(* PLC project Adressering.ecp, WAGO e!COCKPIT e!COCKPIT *)
(* stored: creationDateTime 2021-01-18T14:20:23.2110188, modificationDateTime 2021-01-18T11:51:27.6823754 *)

{attribute 'qualified_only'}
VAR_GLOBAL  (* STLV80_563 *)
  STLV80_A_563_5A201 : dtRomtype_1;  (* Gang *)
  STLV80_A_563_5A202 : dtRomtype_11;  (* gang *)
  STLV80_A_563_5A203 : dtRomtype_111;  (* rom *)
  STLV80_A_563_5A301 : dtRomtype_1111;  (* rom2 *)
  STLV80_A_563_5A302 : dtRomtype_11111;  (* rom3 *)
  STLV80_A_563_5B201 : dtRomtype_111111;  (* rom4 *)
  STLV80_A_563_5B202 : dtRomtype_1111111;  (* rom5 *)
  STLV80_A_563_5B301 : dtRomtype_11111111;  (* rom6 *)
  STLV80_A_563_5B302 : dtRomtype_1111111111;  (* rom7 *)
  STLV80_A_563_5C201 : dtRomtype_1100000001;  (* rom8 *)
  STLV80_A_563_5C202 : dtRomtype_1100000010;  (* 1100000010 *)
END_VAR

PROGRAM PRG_563_KNX
  VAR
    i : INT := 0;  (* Felles *)
    Interval : OSCAT_BASIC.CLK_PRG;
    typDPT : typDPT;
    M1_001_5A201_RB601_V : fbDPT_Switch_pro;  (* 5A201 *)
    M1_002_5A202_RB601_V : fbDPT_Switch_pro;  (* 5A202 *)
    M1_003_5A202_RB601_HVAC : fbDPT_Switch_pro;  (* 5A202 *)
    M1_004_5A203_RB601_V : fbDPT_Switch_pro;  (* 5A203 *)
    M1_005_5A203_RB601_HVAC : fbDPT_Switch_pro;  (* 5A203 *)
    M1_006_5A203_RT601_CT : fbDPT_Value_Temp_pro;  (* 5A203 *)
    M1_007_5A301_RB601_V : fbDPT_Switch_pro;  (* 5A301 *)
    M1_008_5A301_RB601_HVAC : fbDPT_Switch_pro;  (* 5A301 *)
    M1_009_5A301_RT601_CT : fbDPT_Value_Temp_pro;  (* 5A301 *)
    M1_010_5A301_RY601_CV : fbDPT_Value_AirQuality_pro;  (* 5A301 *)
    M1_011_5A302_RB601_V : fbDPT_Switch_pro;  (* 5A302 *)
    M1_012_5A302_RB601_HVAC : fbDPT_Switch_pro;  (* 5A302 *)
    M1_013_5A302_RT601_CT : fbDPT_Value_Temp_pro;  (* 5A302 *)
    M1_014_5A302_RY601_CV : fbDPT_Value_AirQuality_pro;  (* 5A302 *)
    M1_015_5A302_LH601_OP : fbDPT_Scaling_pro;  (* 5A302 *)
    M1_016_5B201_RB601_V : fbDPT_Switch_pro;  (* 5B201 *)
    M1_017_5B201_RB601_HVAC : fbDPT_Switch_pro;  (* 5B201 *)
    M1_018_5B201_RT601_CT : fbDPT_Value_Temp_pro;  (* 5B201 *)
    M1_019_5B201_RY601_CV : fbDPT_Value_AirQuality_pro;  (* 5B201 *)
    M1_020_5B201_LH601_OP : fbDPT_Scaling_pro;  (* 5B201 *)
    M1_021_5B201_LH601_CMD : fbDPT_Switch_pro;  (* 5B201 *)
    M1_022_5B202_RB601_V : fbDPT_Switch_pro;  (* 5B202 *)
    M1_023_5B202_RB601_HVAC : fbDPT_Switch_pro;  (* 5B202 *)
    M1_024_5B202_RT601_CT : fbDPT_Value_Temp_pro;  (* 5B202 *)
    M1_025_5B202_RY601_CV : fbDPT_Value_AirQuality_pro;  (* 5B202 *)
    M1_026_5B202_LH601_OP : fbDPT_Scaling_pro;  (* 5B202 *)
    M1_027_5B202_LH601_CMD : fbDPT_Switch_pro;  (* 5B202 *)
    M1_028_5B202_LC601_OP : fbDPT_Scaling_pro;  (* 5B202 *)
    M1_029_5B301_RB601_V : fbDPT_Switch_pro;  (* 5B301 *)
    M1_030_5B301_RB601_HVAC : fbDPT_Switch_pro;  (* 5B301 *)
    M1_031_5B301_RT601_CT : fbDPT_Value_Temp_pro;  (* 5B301 *)
    M1_032_5B301_RY601_CV : fbDPT_Value_AirQuality_pro;  (* 5B301 *)
    M1_033_5B301_LH601_OP : fbDPT_Scaling_pro;  (* 5B301 *)
    M1_034_5B301_LH601_CMD : fbDPT_Switch_pro;  (* 5B301 *)
    M1_035_5B301_LC601_OP : fbDPT_Scaling_pro;  (* 5B301 *)
    M1_036_5B301_LC601_CMD : fbDPT_Switch_pro;  (* 5B301 *)
    M1_037_5B302_RB601_V : fbDPT_Switch_pro;  (* 5B302 *)
    M1_038_5B302_RB601_HVAC : fbDPT_Switch_pro;  (* 5B302 *)
    M1_039_5B302_RT601_CT : fbDPT_Value_Temp_pro;  (* 5B302 *)
    M1_040_5B302_RY601_CV : fbDPT_Value_AirQuality_pro;  (* 5B302 *)
    M1_041_5B302_LH601_OP : fbDPT_Scaling_pro;  (* 5B302 *)
    M1_042_5B302_LH601_CMD : fbDPT_Switch_pro;  (* 5B302 *)
    M1_043_5B302_LC601_OP : fbDPT_Scaling_pro;  (* 5B302 *)
    M1_044_5B302_LC601_CMD : fbDPT_Switch_pro;  (* 5B302 *)
    M1_045_5B302_RT601_SP_FB : fbDPT_Value_Temp_pro;  (* 5B302 *)
    M1_046_5B302_RT601_SP : fbDPT_Value_Temp_pro;  (* 5B302 *)
    M1_047_5C201_RB601_V : fbDPT_Switch_pro;  (* 5C201 *)
    M1_048_5C201_RB601_HVAC : fbDPT_Switch_pro;  (* 5C201 *)
    M1_049_5C201_RT601_SP : fbDPT_Value_Temp_pro;  (* 5C201 *)
    M1_050_5C202_RB601_V : fbDPT_Switch_pro;  (* 5C202 *)
    M1_051_5C202_RB601_HVAC : fbDPT_Switch_pro;  (* 5C202 *)
    M1_052_5C202_RT601_SP_FB : fbDPT_Value_Temp_pro;  (* 5C202 *)
  END_VAR
  VAR  (* added by the conversion: wires and edge detectors of the diagram *)
    _ADD9_OUT : INT;
    _GT15_OUT : BOOL;
    _MOVE19_ENO : BOOL;
    _MOVE19_OUT : INT;
  END_VAR

(* CFC diagram, written out as Structured Text *)
(* KNX Sending interval *)
Interval(PT := t#2M);
_ADD9_OUT := BOOL_TO_INT(Interval.Q) + i;
i := _ADD9_OUT;
_GT15_OUT := i > 13;
_MOVE19_OUT := MOVE(EN := _GT15_OUT, IN := 0, ENO => _MOVE19_ENO);
IF _MOVE19_ENO THEN i := _MOVE19_OUT; END_IF;
(* Rom 5A201 *)
(* RB601_V *)
M1_001_5A201_RB601_V(bPortKNX := 1, dwIndex_DPT := 1, typDPT := typDPT);
STLV80_563.STLV80_A_563_5A201.RB601_V := M1_001_5A201_RB601_V.xSwitch_OUT;
(* Rom 5A202 *)
(* RB601_V *)
(* RB601_HVAC *)
M1_002_5A202_RB601_V(bPortKNX := 1, dwIndex_DPT := 2, typDPT := typDPT);
STLV80_563.STLV80_A_563_5A202.RB601_V := M1_002_5A202_RB601_V.xSwitch_OUT;
M1_003_5A202_RB601_HVAC(bPortKNX := 1, dwIndex_DPT := 3, typDPT := typDPT);
STLV80_563.STLV80_A_563_5A202.RB601_HVAC := M1_003_5A202_RB601_HVAC.xSwitch_OUT;
(* Rom 5A203 *)
(* RB601_V *)
(* RB601_HVAC *)
M1_004_5A203_RB601_V(bPortKNX := 1, dwIndex_DPT := 4, typDPT := typDPT);
STLV80_563.STLV80_A_563_5A203.RB601_V := M1_004_5A203_RB601_V.xSwitch_OUT;
M1_005_5A203_RB601_HVAC(bPortKNX := 1, dwIndex_DPT := 5, typDPT := typDPT);
STLV80_563.STLV80_A_563_5A203.RB601_HVAC := M1_005_5A203_RB601_HVAC.xSwitch_OUT;
(* RT601_CT *)
M1_006_5A203_RT601_CT(bPortKNX := 1, dwIndex_DPT := 6, typDPT := typDPT);
STLV80_563.STLV80_A_563_5A203.RT601_CT := M1_006_5A203_RT601_CT.rValue_OUT;
(* Rom 5A301 *)
(* RB601_V *)
(* RB601_HVAC *)
M1_007_5A301_RB601_V(bPortKNX := 1, dwIndex_DPT := 7, typDPT := typDPT);
STLV80_563.STLV80_A_563_5A301.RB601_V := M1_007_5A301_RB601_V.xSwitch_OUT;
M1_008_5A301_RB601_HVAC(bPortKNX := 1, dwIndex_DPT := 8, typDPT := typDPT);
STLV80_563.STLV80_A_563_5A301.RB601_HVAC := M1_008_5A301_RB601_HVAC.xSwitch_OUT;
(* RT601_CT *)
(* RY601_CV *)
M1_009_5A301_RT601_CT(bPortKNX := 1, dwIndex_DPT := 9, typDPT := typDPT);
STLV80_563.STLV80_A_563_5A301.RT601_CT := M1_009_5A301_RT601_CT.rValue_OUT;
M1_010_5A301_RY601_CV(bPortKNX := 1, dwIndex_DPT := 10, typDPT := typDPT);
STLV80_563.STLV80_A_563_5A301.RY601_CV := M1_010_5A301_RY601_CV.rValue_OUT;
(* Rom 5A302 *)
(* RB601_V *)
(* RB601_HVAC *)
M1_011_5A302_RB601_V(bPortKNX := 1, dwIndex_DPT := 11, typDPT := typDPT);
STLV80_563.STLV80_A_563_5A302.RB601_V := M1_011_5A302_RB601_V.xSwitch_OUT;
M1_012_5A302_RB601_HVAC(bPortKNX := 1, dwIndex_DPT := 12, typDPT := typDPT);
STLV80_563.STLV80_A_563_5A302.RB601_HVAC := M1_012_5A302_RB601_HVAC.xSwitch_OUT;
(* RT601_CT *)
(* RY601_CV *)
M1_013_5A302_RT601_CT(bPortKNX := 1, dwIndex_DPT := 13, typDPT := typDPT);
STLV80_563.STLV80_A_563_5A302.RT601_CT := M1_013_5A302_RT601_CT.rValue_OUT;
M1_014_5A302_RY601_CV(bPortKNX := 1, dwIndex_DPT := 14, typDPT := typDPT);
STLV80_563.STLV80_A_563_5A302.RY601_CV := M1_014_5A302_RY601_CV.rValue_OUT;
(* LH601_OP *)
M1_015_5A302_LH601_OP(bPortKNX := 1, dwIndex_DPT := 15, rValue_IN := STLV80_563.STLV80_A_563_5A302.LH601_OP, xUpdate_KNX := i = 0, typDPT := typDPT);
(* Rom 5B201 *)
(* RB601_V *)
(* RB601_HVAC *)
M1_016_5B201_RB601_V(bPortKNX := 1, dwIndex_DPT := 16, typDPT := typDPT);
STLV80_563.STLV80_A_563_5B201.RB601_V := M1_016_5B201_RB601_V.xSwitch_OUT;
M1_017_5B201_RB601_HVAC(bPortKNX := 1, dwIndex_DPT := 17, typDPT := typDPT);
STLV80_563.STLV80_A_563_5B201.RB601_HVAC := M1_017_5B201_RB601_HVAC.xSwitch_OUT;
(* RT601_CT *)
(* RY601_CV *)
M1_018_5B201_RT601_CT(bPortKNX := 1, dwIndex_DPT := 18, typDPT := typDPT);
STLV80_563.STLV80_A_563_5B201.RT601_CT := M1_018_5B201_RT601_CT.rValue_OUT;
M1_019_5B201_RY601_CV(bPortKNX := 1, dwIndex_DPT := 19, typDPT := typDPT);
STLV80_563.STLV80_A_563_5B201.RY601_CV := M1_019_5B201_RY601_CV.rValue_OUT;
(* LH601_OP *)
(* LH601_CMD *)
M1_020_5B201_LH601_OP(bPortKNX := 1, dwIndex_DPT := 20, rValue_IN := STLV80_563.STLV80_A_563_5B201.LH601_OP, xUpdate_KNX := i = 1, typDPT := typDPT);
M1_021_5B201_LH601_CMD(bPortKNX := 1, dwIndex_DPT := 21, xSwitch_IN := STLV80_563.STLV80_A_563_5B201.LH601_CMD, xUpdate_KNX := i = 2, typDPT := typDPT);
(* Rom 5B202 *)
(* RB601_V *)
(* RB601_HVAC *)
M1_022_5B202_RB601_V(bPortKNX := 1, dwIndex_DPT := 22, typDPT := typDPT);
STLV80_563.STLV80_A_563_5B202.RB601_V := M1_022_5B202_RB601_V.xSwitch_OUT;
M1_023_5B202_RB601_HVAC(bPortKNX := 1, dwIndex_DPT := 23, typDPT := typDPT);
STLV80_563.STLV80_A_563_5B202.RB601_HVAC := M1_023_5B202_RB601_HVAC.xSwitch_OUT;
(* RT601_CT *)
(* RY601_CV *)
M1_024_5B202_RT601_CT(bPortKNX := 1, dwIndex_DPT := 24, typDPT := typDPT);
STLV80_563.STLV80_A_563_5B202.RT601_CT := M1_024_5B202_RT601_CT.rValue_OUT;
M1_025_5B202_RY601_CV(bPortKNX := 1, dwIndex_DPT := 25, typDPT := typDPT);
STLV80_563.STLV80_A_563_5B202.RY601_CV := M1_025_5B202_RY601_CV.rValue_OUT;
(* LH601_OP *)
(* LH601_CMD *)
M1_026_5B202_LH601_OP(bPortKNX := 1, dwIndex_DPT := 26, rValue_IN := STLV80_563.STLV80_A_563_5B202.LH601_OP, xUpdate_KNX := i = 3, typDPT := typDPT);
M1_027_5B202_LH601_CMD(bPortKNX := 1, dwIndex_DPT := 27, xSwitch_IN := STLV80_563.STLV80_A_563_5B202.LH601_CMD, xUpdate_KNX := i = 4, typDPT := typDPT);
(* LC601_OP *)
M1_028_5B202_LC601_OP(bPortKNX := 1, dwIndex_DPT := 28, rValue_IN := STLV80_563.STLV80_A_563_5B202.LC601_OP, xUpdate_KNX := i = 5, typDPT := typDPT);
(* Rom 5B301 *)
(* RB601_V *)
(* RB601_HVAC *)
M1_029_5B301_RB601_V(bPortKNX := 1, dwIndex_DPT := 29, typDPT := typDPT);
STLV80_563.STLV80_A_563_5B301.RB601_V := M1_029_5B301_RB601_V.xSwitch_OUT;
M1_030_5B301_RB601_HVAC(bPortKNX := 1, dwIndex_DPT := 30, typDPT := typDPT);
STLV80_563.STLV80_A_563_5B301.RB601_HVAC := M1_030_5B301_RB601_HVAC.xSwitch_OUT;
(* RT601_CT *)
(* RY601_CV *)
M1_031_5B301_RT601_CT(bPortKNX := 1, dwIndex_DPT := 31, typDPT := typDPT);
STLV80_563.STLV80_A_563_5B301.RT601_CT := M1_031_5B301_RT601_CT.rValue_OUT;
M1_032_5B301_RY601_CV(bPortKNX := 1, dwIndex_DPT := 32, typDPT := typDPT);
STLV80_563.STLV80_A_563_5B301.RY601_CV := M1_032_5B301_RY601_CV.rValue_OUT;
(* LH601_OP *)
(* LH601_CMD *)
M1_033_5B301_LH601_OP(bPortKNX := 1, dwIndex_DPT := 33, rValue_IN := STLV80_563.STLV80_A_563_5B301.LH601_OP, xUpdate_KNX := i = 6, typDPT := typDPT);
M1_034_5B301_LH601_CMD(bPortKNX := 1, dwIndex_DPT := 34, xSwitch_IN := STLV80_563.STLV80_A_563_5B301.LH601_CMD, xUpdate_KNX := i = 7, typDPT := typDPT);
(* LC601_OP *)
(* LC601_CMD *)
M1_035_5B301_LC601_OP(bPortKNX := 1, dwIndex_DPT := 35, rValue_IN := STLV80_563.STLV80_A_563_5B301.LC601_OP, xUpdate_KNX := i = 8, typDPT := typDPT);
M1_036_5B301_LC601_CMD(bPortKNX := 1, dwIndex_DPT := 36, xSwitch_IN := STLV80_563.STLV80_A_563_5B301.LC601_CMD, xUpdate_KNX := i = 9, typDPT := typDPT);
(* Rom 5B302 *)
(* RB601_V *)
(* RB601_HVAC *)
M1_037_5B302_RB601_V(bPortKNX := 1, dwIndex_DPT := 37, typDPT := typDPT);
STLV80_563.STLV80_A_563_5B302.RB601_V := M1_037_5B302_RB601_V.xSwitch_OUT;
M1_038_5B302_RB601_HVAC(bPortKNX := 1, dwIndex_DPT := 38, typDPT := typDPT);
STLV80_563.STLV80_A_563_5B302.RB601_HVAC := M1_038_5B302_RB601_HVAC.xSwitch_OUT;
(* RT601_CT *)
(* RY601_CV *)
M1_039_5B302_RT601_CT(bPortKNX := 1, dwIndex_DPT := 39, typDPT := typDPT);
STLV80_563.STLV80_A_563_5B302.RT601_CT := M1_039_5B302_RT601_CT.rValue_OUT;
M1_040_5B302_RY601_CV(bPortKNX := 1, dwIndex_DPT := 40, typDPT := typDPT);
STLV80_563.STLV80_A_563_5B302.RY601_CV := M1_040_5B302_RY601_CV.rValue_OUT;
(* LH601_OP *)
(* LH601_CMD *)
M1_041_5B302_LH601_OP(bPortKNX := 1, dwIndex_DPT := 41, rValue_IN := STLV80_563.STLV80_A_563_5B302.LH601_OP, xUpdate_KNX := i = 10, typDPT := typDPT);
M1_042_5B302_LH601_CMD(bPortKNX := 1, dwIndex_DPT := 42, xSwitch_IN := STLV80_563.STLV80_A_563_5B302.LH601_CMD, xUpdate_KNX := i = 11, typDPT := typDPT);
(* LC601_OP *)
(* LC601_CMD *)
M1_043_5B302_LC601_OP(bPortKNX := 1, dwIndex_DPT := 43, rValue_IN := STLV80_563.STLV80_A_563_5B302.LC601_OP, xUpdate_KNX := i = 12, typDPT := typDPT);
M1_044_5B302_LC601_CMD(bPortKNX := 1, dwIndex_DPT := 44, xSwitch_IN := STLV80_563.STLV80_A_563_5B302.LC601_CMD, xUpdate_KNX := i = 13, typDPT := typDPT);
(* RT601_SP *)
(* RT601_SP Feedback *)
M1_045_5B302_RT601_SP(bPortKNX := 1, dwIndex_DPT := 45, rValue_IN := STLV80_563.STLV80_A_563_5B302.RT601_SP_D, xUpdate_KNX := NOT STLV80_563.STLV80_A_563_5B302.RB601_HVAC, typDPT := typDPT);
M1_046_5B302_RT601_SP_FB(bPortKNX := 1, dwIndex_DPT := 46, typDPT := typDPT);
STLV80_563.STLV80_A_563_5B302.RT601_SP_IN := M1_046_5B302_RT601_SP_FB.rValue_OUT;
(* Rom 5C201 *)
(* RB601_V *)
(* RB601_HVAC *)
M1_047_5C201_RB601_V(bPortKNX := 1, dwIndex_DPT := 47, typDPT := typDPT);
STLV80_563.STLV80_A_563_5C201.RB601_V := M1_047_5C201_RB601_V.xSwitch_OUT;
M1_048_5C201_RB601_HVAC(bPortKNX := 1, dwIndex_DPT := 48, typDPT := typDPT);
STLV80_563.STLV80_A_563_5C201.RB601_HVAC := M1_048_5C201_RB601_HVAC.xSwitch_OUT;
(* RT601_SP Feedback *)
M1_049_5C201_RT601_SP_FB(bPortKNX := 1, dwIndex_DPT := 49, typDPT := typDPT);
STLV80_563.STLV80_A_563_5C201.RT601_SP_IN := M1_049_5C201_RT601_SP_FB.rValue_OUT;
(* Rom 5C202 *)
(* RB601_V *)
(* RB601_HVAC *)
M1_050_5C202_RB601_V(bPortKNX := 1, dwIndex_DPT := 50, typDPT := typDPT);
STLV80_563.STLV80_A_563_5C202.RB601_V := M1_050_5C202_RB601_V.xSwitch_OUT;
M1_051_5C202_RB601_HVAC(bPortKNX := 1, dwIndex_DPT := 51, typDPT := typDPT);
STLV80_563.STLV80_A_563_5C202.RB601_HVAC := M1_051_5C202_RB601_HVAC.xSwitch_OUT;
(* RT601_SP *)
M1_052_5C202_RT601_SP(bPortKNX := 1, dwIndex_DPT := 52, rValue_IN := STLV80_563.STLV80_A_563_5C202.RT601_SP_D, xUpdate_KNX := NOT STLV80_563.STLV80_A_563_5C202.RB601_HVAC, typDPT := typDPT);
END_PROGRAM
